// TIA Portal V17 export
// export: Created 2025-04-05T13:39:33.1172665Z, ExportSetting WithDefaults, DisplayName Totally Integrated Automation Portal, DisplayVersion V17, DisplayName TIA Portal Openness, DisplayVersion V17, DisplayName TIA Portal Version Control Interface, DisplayVersion V17, DisplayName STEP 7 Professional, DisplayVersion V17, DisplayName STEP 7 Safety, DisplayVersion V17, DisplayName WinCC Advanced, DisplayVersion V17
VAR_GLOBAL   // PLC tag table "DI"
   I0 AT %I20.0 : Bool;
   I1 AT %I20.1 : Bool;
   I2 AT %I20.2 : Bool;
   I3 AT %I20.3 : Bool;
   I4 AT %I20.4 : Bool;
   I5 AT %I20.5 : Bool;
   I6 AT %I20.6 : Bool;
   I7 AT %I20.7 : Bool;
   I8 AT %I21.0 : Bool;
   I9 AT %I21.1 : Bool;
   I10 AT %I21.2 : Bool;
   I11 AT %I21.3 : Bool;
   I12 AT %I21.4 : Bool;
   I13 AT %I21.5 : Bool;
   I14 AT %I21.6 : Bool;
   I15 AT %I21.7 : Bool;
   I16 AT %I22.0 : Bool;
   I17 AT %I22.1 : Bool;
   I18 AT %I22.2 : Bool;
   I19 AT %I22.3 : Bool;
   I20 AT %I22.4 : Bool;
   I21 AT %I22.5 : Bool;
   I22 AT %I22.6 : Bool;
   I23 AT %I22.7 : Bool;
   I24 AT %I23.0 : Bool;
   I25 AT %I23.1 : Bool;
   I26 AT %I23.2 : Bool;
   I27 AT %I23.3 : Bool;
   I28 AT %I23.4 : Bool;
   I29 AT %I23.5 : Bool;
   I30 AT %I23.6 : Bool;
   I31 AT %I23.7 : Bool;
   Tag_1 AT %IW26 : Word;
   Tag_2 AT %IW24 : Word;
   Tag_3 AT %IW22 : Word;
END_VAR
